// TwinCAT 3 PLC project plc
// ProgramVersion: 3.1.4024.0
// libraries:
//   Tc2_Standard, * (Beckhoff Automation GmbH)
//   Tc2_System, * (Beckhoff Automation GmbH)
//   Tc3_Module, * (Beckhoff Automation GmbH)
// project tree:
//   GVLs/ GVL.TcGVL
//   / PlcTask.TcTTO
//   POUs/ MAIN.TcPOU
// real-time tasks:
//   TASK PlcTask: cycle T#10ms, priority 20, ADS port 350

CONFIGURATION plc
    RESOURCE PLC ON TwinCAT3
        TASK PlcTask(INTERVAL := T#10ms, PRIORITY := 20);
        PROGRAM MAIN WITH PlcTask : MAIN;
    END_RESOURCE
END_CONFIGURATION

// ---- GVLs/GVL.TcGVL
{attribute 'qualified_only'}
VAR_GLOBAL
	

  rX 			: REAL;
  rY			: REAL;
  iA			: INT;
  
  //mootor controls 
  
  bmotorstartpb 	: BOOL;
  bmotorstoppb		: BOOL;
  bmotorcontrol		: BOOL;
  
  bmotorcontrolenable : BOOL;
  
  
END_VAR

// ---- POUs/MAIN.TcPOU
PROGRAM MAIN
VAR
END_VAR

M_SING();
M_MOTOR();

METHOD M_MOTOR : BOOL
VAR_INPUT
END_VAR
gvl.bmotorcontrol := ((gvl.bmotorstartpb or gvl.bmotorcontrol) and (not gvl.bmotorstoppb) ) and gvl.bmotorcontrolenable;

//	GVL.bmotorstartpb := false;
//	gvl.bmotorstoppb := false;
END_METHOD

METHOD M_SING : BOOL
VAR_INPUT
END_VAR


GVL.RX 		:= 0.02 + GVL.rX;

IF GVL.rY > (3.14 * 2.0) THEN
	
	GVL.RX := 0;
	
END_IF
GVL.rY  	:= SIN(GVL.RX);
END_METHOD

END_PROGRAM
